FUNCTION_BLOCK CurtainWithSensor EXTENDS Curtain
VAR
	OpenSensor	AT%I* : BOOL;
	CloseSensor	AT%I* : BOOL;

	_OpeningTime: TIME;
	_ClosingTime: TIME;
	_status: REAL;

	M_CalibrationAttempt_open: BOOL;
	M_CalibrationAttempt_close: BOOL;
	tonOpenTimeMeasurement: TON;
	tonCloseTimeMeasurement: TON;
	tonStatusTracker_open: TON;
	tonStatusTracker_close: TON;
	statusTrackerTime: TIME;
	rtIN_open: BOOL;
	rtIN_close: BOOL;
END_VAR

METHOD Close : BOOL
VAR_INPUT
	IN: BOOL;
END_VAR

//	Status - Travel time Calibration (Close Time)
IF OpenSensor AND IN THEN
	M_CalibrationAttempt_close	:=	TRUE;
	tonCloseTimeMeasurement(IN:= FALSE, PT:= T#1D, Q=> , ET=> );
END_IF
IF M_CalibrationAttempt_close AND (NOT OpenSensor) THEN
	toncloseTimeMeasurement(IN:= TRUE, PT:= T#1D, Q=> , ET=> );
END_IF


IF NOT Open_op THEN
	Close_op	:=	IN;

	IF NOT rtIN_close THEN
		rtIN_close			:=	TRUE;		
		statusTrackerTime	:=	REAL_TO_TIME(F_Scaling(Variable_In:= _status, Input_min:= 0, Input_max:= 100, Output_min:= 0, Output_max:= TIME_TO_REAL(_ClosingTime)));			
	END_IF

	tonStatusTracker_close(IN:= close_op, PT:= _closingTime, Q=> , ET=> );
	IF tonStatusTracker_close.IN THEN
		IF statusTrackerTime >= tonStatusTracker_close.ET THEN
			_status	:=	LIMIT( 0, (F_Scaling(Variable_In:= TIME_TO_REAL(statusTrackerTime - tonStatusTracker_close.ET), Input_min:= 0, Input_max:= TIME_TO_REAL(_closingTime), Output_min:= 0, Output_max:= 100)) , 100);
		ELSE
			_status	:=	0;	
		END_IF			
	END_IF
	
END_IF

IF CloseSensor THEN
	Close_op	:=	FALSE;
	
	IF M_CalibrationAttempt_close AND (NOT OpenSensor) THEN
		M_CalibrationAttempt_close	:=	FALSE;
		_ClosingTime			:=	toncloseTimeMeasurement.ET;
		toncloseTimeMeasurement(IN:= FALSE, PT:= T#1D, Q=> , ET=> );
		_status					:=	0;
	END_IF
END_IF

IF (IN = FALSE) THEN
	M_CalibrationAttempt_close	:=	FALSE;
	toncloseTimeMeasurement(IN:= FALSE, PT:= T#1D, Q=> , ET=> );
	tonStatusTracker_close(IN:= FALSE, PT:= , Q=> , ET=> );
	rtIN_close	:=	FALSE;	
END_IF
	
toncloseTimeMeasurement();
tonStatusTracker_close();
END_METHOD

METHOD Open : BOOL
VAR_INPUT
	IN: BOOL;
END_VAR

//	Status - Travel time Calibration (Open Time)
IF CloseSensor AND IN THEN
	M_CalibrationAttempt_open	:=	TRUE;
	tonOpenTimeMeasurement(IN:= FALSE, PT:= T#1D, Q=> , ET=> );
END_IF
IF M_CalibrationAttempt_open AND (NOT CloseSensor) THEN
	tonOpenTimeMeasurement(IN:= TRUE, PT:= T#1D, Q=> , ET=> );
END_IF


IF NOT Close_op THEN
	Open_op	:=	IN;
	
	IF NOT rtIN_open THEN
		rtIN_open			:=	TRUE;
		statusTrackerTime	:=	REAL_TO_TIME(F_Scaling(Variable_In:= _status, Input_min:= 0, Input_max:= 100, Output_min:= 0, Output_max:= TIME_TO_REAL(_OpeningTime)));			
	END_IF

	tonStatusTracker_open(IN:= Open_op, PT:= _OpeningTime, Q=> , ET=> );
	IF tonStatusTracker_open.IN THEN
		IF (tonStatusTracker_open.ET <= _OpeningTime) THEN
			_status	:=	LIMIT( 0, F_Scaling(Variable_In:= TIME_TO_REAL(statusTrackerTime + tonStatusTracker_open.ET), Input_min:= 0, Input_max:= TIME_TO_REAL(_OpeningTime), Output_min:= 0, Output_max:= 100), 100);
		ELSE
			_status	:=	100;	
		END_IF			
	END_IF
		
END_IF

IF OpenSensor THEN
	Open_op	:=	FALSE;
	
	IF M_CalibrationAttempt_open AND (NOT CloseSensor) THEN
		M_CalibrationAttempt_open	:=	FALSE;
		_OpeningTime			:=	tonOpenTimeMeasurement.ET;
		tonOpenTimeMeasurement(IN:= FALSE, PT:= T#1D, Q=> , ET=> );
		_status					:=	100;
	END_IF
END_IF

IF (IN = FALSE) THEN
	M_CalibrationAttempt_open	:=	FALSE;
	tonOpenTimeMeasurement(IN:= FALSE, PT:= T#1D, Q=> , ET=> );
	tonStatusTracker_open(IN:= FALSE, PT:= , Q=> , ET=> );
	rtIN_open	:=	FALSE;
END_IF
	
tonOpenTimeMeasurement();
tonStatusTracker_open();
END_METHOD

PROPERTY Status : INT
GET
Status	:=	REAL_TO_INT(_status);
END_GET
END_PROPERTY

END_FUNCTION_BLOCK

(* stored: Version 1.1.0.1, ProductVersion 3.1.4024.13
   POU CurtainWithSensor: Id {966f90ac-e61b-44c1-9f86-ea4c94f38c65}, SpecialFunc None
   Method Close: Id {1ea6e25f-e983-4dbe-ba01-81447cc68a62}
   Method Open: Id {611fa041-c933-4221-b71b-b0e5334120fb}
   Property Status: Id {43526895-7814-462c-8028-3821f4aa44c0}
   Get Get: Id {640bccd9-ad01-4a1c-a206-7522b59a5002} *)
